(* CODESYS project ringbuffer.library
   Author: vscottki
   Placeholder: RingBuffer
   Title: RingBuffer
   Version: 1.4.0.999
   Company: Amazon

Project tree, tasks and I/O mapping:
  libraries: HelperFunctions, * (Amazon); Tc2_Standard, * (Beckhoff Automation GmbH); Tc2_System, * (Beckhoff Automation GmbH); Tc3_Module, * (Beckhoff Automation GmbH)
  DUTs/
    data type E_Divert
    data type ST_KeyValue
    data type ST_MoverDivert
    data type ST_RingBufferCfg
    data type ST_RingBufferStat
    data type ST_SystimeString
  GVLs/
    global variables Param_RingBuffer
  POUs/
    function block RingBufferBase [ST]: UpdateObjectCtInBuffers, P_ObjCountInBuffer, P_ObjectAdded, P_ObjectRemoved, ClearLastRemoved, IncrementPointer, UpdateAdded, UpdateIndices, UpdateRemoved, UpdateRemovePointer, UpdateWritePointer, FB_init
    function block RingBufferEventBase [ST]: ClearLastRemoved, UpdateRemovePointer, UpdateWritePointer, AddObjToBuffer, FB_init, P_LastObjectRemoved, RemoveObjFromBuffer, EqualsTo, EqualsToEventClass, EqualsToEventEntry, EqualsToEventEntryEx, eSeverity, EventClass, GetJsonAttribute, ipSourceInfo, nEventId, RequestEventClassName, RequestEventText, sEventClassName, sEventText, stEventEntry
    function block RingBufferKeyString [ST]: ClearLastRemoved, UpdateRemovePointer, UpdateWritePointer, AddObjToBuffer, FB_init, P_LastObjectRemoved, RemoveObjFromBuffer, CopyMemArea
    function block RingBufferMoverDivert [ST]: ClearLastRemoved, UpdateRemovePointer, UpdateWritePointer, AddObjToBuffer, FB_init, P_LastObjectRemoved, RemoveObjFromBuffer
    function UpdateKeyStrTimestamp [ST]
    function UpdateKeyValueTimestamp [ST]
  Project Information/
    function F_GetCompany [ST]
    function F_GetTitle [ST]
    function F_GetVersion [ST]
  Version/
    global variables Global_Version
  VISUs/
*)

// DUTs/E_Divert
{attribute 'qualified_only'}
{attribute 'strict'}
TYPE E_Divert :
(
	NoDivert := 0,
	Divert	:= 1
);
END_TYPE

// DUTs/ST_KeyValue
TYPE ST_KeyValue :
STRUCT
  key         : ULINT;    // system timestamp
  value       : ULINT; // SJsonValue;+ dynamically spool up instances of JSONDOMparser to create documents, then destroy them when completed; 
END_STRUCT
END_TYPE

// DUTs/ST_MoverDivert
TYPE ST_MoverDivert :
STRUCT
	MoverID						: UDINT;
	Divert						: E_Divert;
	DivertOnInterval	: BOOL;
	SysTime     			: ULINT;    // system timestamp
END_STRUCT
END_TYPE

// DUTs/ST_RingBufferCfg
TYPE ST_RingBufferCfg :
STRUCT
  CopyToLargeMemoryArea   : BOOL := TRUE;
  CopyOnlyUniqueMessage   : BOOL := FALSE;
  AllowOverwriteSecBuffer : BOOL := FALSE;
  ByteCountOfDataObj      : UDINT; // do not write to this manually; done using SIZEOF function
  WriteDataToFile         : BOOL := FALSE;
	RemoveAfterAdd					: BOOL;
END_STRUCT
END_TYPE

// DUTs/ST_RingBufferStat
TYPE ST_RingBufferStat :
STRUCT
  BufferIsFullPrim        : BOOL;
  BufferIsFullSec         : BOOL;  
  ObjectCountInBufferPrim : ULINT;
  ObjectCountInBufferSec  : ULINT;
  ObjectAddedPrimary      : BOOL;
  ObjectRemovedPrimary    : BOOL;
  ObjectAdded2ndary       : BOOL;
  ObjectRemoved2ndary     : BOOL;
  Overwriting             : BOOL;
  ByteCountInBufferPrim   : ULINT;  
  ByteCountInBufferSec    : ULINT;
  BufferCapacity          : UDINT;
END_STRUCT
END_TYPE

// DUTs/ST_SystimeString
TYPE ST_SystimeString :
STRUCT
  systimestamp   : ULINT;    // system timestamp
  sJson          : TcEventField.JsonAttribute;
  stringval      : Tc2_System.T_MaxString;
END_STRUCT
END_TYPE

// GVLs/Param_RingBuffer
{attribute 'qualified_only'}
VAR_GLOBAL CONSTANT
  MIN_NUMBER_OBJECTS : UDINT := 0;
  MAX_NUMBER_OBJECTS : UDINT := 4;
END_VAR

// Version/Global_Version
{attribute 'TcGenerated'}
{attribute 'no-analysis'}
{attribute 'linkalways'}
// This function has been automatically generated from the project information.
VAR_GLOBAL CONSTANT
	{attribute 'const_non_replaced'}
	stLibVersion_RingBuffer : ST_LibVersion := (iMajor := 1, iMinor := 4, iBuild := 0, iRevision := 999, nFlags := 0, sVersion := '1.4.0.999');
END_VAR

// POUs/RingBufferBase
FUNCTION_BLOCK ABSTRACT RingBufferBase
VAR
  RingBuffCfg             : ST_RingBufferCfg;
  pRemove                 : PVOID;
  pWrite                  : PVOID;
  pRemoveUpdated          : BOOL;
  pWriteUpdated           : BOOL;
  GlobalCounter           : UDINT;
  WriteIncrement          : UDINT;
  RemoveIncrement         : UDINT;
  WriteIndex              : UDINT;
  RemoveIndex             : UDINT;
  RingBufferStat          : ST_RingBufferStat;
END_VAR

UpdateObjectCtInBuffers();
UpdateIndices();

METHOD PRIVATE UpdateObjectCtInBuffers
IF RingBufferStat.ObjectAddedPrimary THEN
  IF GlobalCounter >= RingBufferStat.BufferCapacity THEN // In Buffer Overflow
    RingBufferStat.ObjectCountInBufferPrim   := RingBufferStat.BufferCapacity;
  ELSE
    RingBufferStat.ObjectCountInBufferPrim   := RingBufferStat.ObjectCountInBufferPrim +1;
	END_IF
END_IF

IF RingBufferStat.ObjectRemovedPrimary THEN
  RingBufferStat.ObjectCountInBufferPrim   := RingBufferStat.ObjectCountInBufferPrim -1; 
END_IF

//Primary - Ring
RingBufferStat.BufferIsFullPrim          := RingBufferStat.ObjectCountInBufferPrim = RingBufferStat.BufferCapacity;
                      
RingBufferStat.ByteCountInBufferPrim     := RingBufferStat.ObjectCountInBufferPrim * RingBuffCfg.ByteCountOfDataObj;

//Secondary
RingBufferStat.BufferIsFullSec           := RingBufferStat.ObjectCountInBufferSec = RingBufferStat.BufferCapacity;
                      
RingBufferStat.ByteCountInBufferSec      := RingBufferStat.ObjectCountInBufferSec * RingBuffCfg.ByteCountOfDataObj;
END_METHOD

{attribute 'monitoring' := 'call'}
PROPERTY P_ObjCountInBuffer : ULINT
GET
P_ObjCountInBuffer  := RingBufferStat.ObjectCountInBufferPrim;
END_GET
END_PROPERTY

PROPERTY P_ObjectAdded : REFERENCE TO BOOL
GET
P_ObjectAdded REF= RingBufferStat.ObjectAddedPrimary;
END_GET
END_PROPERTY

PROPERTY P_ObjectRemoved : REFERENCE TO BOOL
GET
P_ObjectRemoved REF= RingBufferStat.ObjectRemovedPrimary;
END_GET
END_PROPERTY

METHOD PROTECTED ABSTRACT ClearLastRemoved
END_METHOD

METHOD PROTECTED IncrementPointer : ULINT
VAR_INPUT
  pPointer        : PVOID;
  ByteCtIncrement : ULINT; 
END_VAR
IncrementPointer  := pPointer + ByteCtIncrement;
END_METHOD

METHOD PROTECTED UpdateAdded
IF RingBufferStat.ObjectAddedPrimary THEN
  RingBufferStat.ObjectAddedPrimary   := FALSE;
END_IF

IF RingBufferStat.ObjectAdded2ndary THEN
  RingBufferStat.ObjectAdded2ndary   := FALSE;
END_IF
END_METHOD

METHOD PROTECTED UpdateIndices
WriteIndex := (WriteIncrement MOD RingBufferStat.BufferCapacity) + Param_RingBuffer.MIN_NUMBER_OBJECTS;

IF GlobalCounter >= RingBufferStat.BufferCapacity THEN // Buffer Overflow
  RemoveIndex                 := WriteIndex+1;
  RingBufferStat.Overwriting  := TRUE;
ELSE
  RemoveIndex  := (RemoveIncrement MOD RingBufferStat.BufferCapacity) + Param_RingBuffer.MIN_NUMBER_OBJECTS;
  RingBufferStat.Overwriting  := FALSE;
END_IF
END_METHOD

METHOD PROTECTED UpdateRemoved
IF RingBufferStat.ObjectRemovedPrimary THEN
  RingBufferStat.ObjectRemovedPrimary   := FALSE;
END_IF

IF RingBufferStat.ObjectRemoved2ndary THEN
  RingBufferStat.ObjectRemoved2ndary   := FALSE;
END_IF
END_METHOD

METHOD PROTECTED ABSTRACT UpdateRemovePointer
VAR_INPUT
  pRemovePtr  : PVOID;
END_VAR
END_METHOD

METHOD PROTECTED ABSTRACT UpdateWritePointer
VAR_INPUT
  pWritePtr  : PVOID;
END_VAR
END_METHOD

METHOD FB_init : BOOL
VAR_INPUT
	bInitRetains : BOOL; // if TRUE, the retain variables are initialized (warm start / cold start)
	bInCopyCode : BOOL;  // if TRUE, the instance afterwards gets moved into the copy code (online change)
END_VAR
RingBufferStat.BufferCapacity  := (Param_RingBuffer.MAX_NUMBER_OBJECTS - Param_RingBuffer.MIN_NUMBER_OBJECTS) +1;
END_METHOD

END_FUNCTION_BLOCK

// POUs/RingBufferEventBase
FUNCTION_BLOCK RingBufferEventBase EXTENDS RingBufferBase
VAR
  Buffer              : ARRAY[Param_RingBuffer.MIN_NUMBER_OBJECTS..Param_RingBuffer.MAX_NUMBER_OBJECTS] 
                        OF ST_KeyValue;
//VAR_OUTPUT
  LastObjRemoved      : ST_KeyValue;
{warning 'Dependency injection from child FB?'}  
//  instQueryInterface  : I_Event := THIS^;//__SYSTEM.IQueryInterface;
END_VAR

SUPER^();

METHOD PROTECTED ClearLastRemoved
IF NOT pRemoveUpdated THEN
  MEMSET(destAddr := ADR(LastObjRemoved), fillByte := 16#00, n := RingBuffCfg.ByteCountOfDataObj);  
END_IF
END_METHOD

METHOD PROTECTED UpdateRemovePointer
VAR_INPUT
  pRemovePtr  : PVOID;
END_VAR
pRemove := ADR(Buffer[RemoveIndex]);

pRemoveUpdated  := TRUE;
END_METHOD

METHOD PROTECTED UpdateWritePointer
VAR_INPUT
  pWritePtr  : PVOID;
END_VAR
IF (WriteIndex = Param_RingBuffer.MIN_NUMBER_OBJECTS) THEN
  pWrite        := ADR(Buffer[Param_RingBuffer.MIN_NUMBER_OBJECTS]);
ELSIF (WriteIndex > Param_RingBuffer.MIN_NUMBER_OBJECTS) AND 
  (WriteIndex <= Param_RingBuffer.MAX_NUMBER_OBJECTS) THEN
  pWrite        := IncrementPointer(pPointer  := pWrite, ByteCtIncrement := RingBuffCfg.ByteCountOfDataObj);
END_IF

pWriteUpdated   := TRUE;
END_METHOD

METHOD PUBLIC AddObjToBuffer
VAR_INPUT
  RefObject           : REFERENCE TO ST_KeyValue;
END_VAR
VAR
  CountBytesWritten   : ULINT;
END_VAR
VAR_OUTPUT
  Error               : BOOL;
END_VAR
UpdateWritePointer(pWritePtr := pWrite);

IF __ISVALIDREF(RefObject) AND pWriteUpdated AND_THEN NOT pRemoveUpdated AND (GlobalCounter < 4294967295) THEN
  UpdateKeyValueTimestamp(DataObject := RefObject);
//  UpdateObjectMemLoc(DataObject := RefObject, _interface := instQueryInterface);
  CountBytesWritten := Tc2_System.MEMMOVE(srcAddr := ADR(RefObject), destAddr := pWrite, n := RingBuffCfg.ByteCountOfDataObj);
  pWriteUpdated     := FALSE;
{warning <'Check Global Buffer Overflow condition if Counter defined > MAX SIZE OF UDINT'>}
END_IF

IF (CountBytesWritten > 0) THEN
  GlobalCounter     := GlobalCounter +1;
  WriteIncrement    := WriteIncrement +1;
  RingBufferStat.ObjectAddedPrimary       := TRUE;
ELSIF (CountBytesWritten <= 0) THEN
  Error             := TRUE;
END_IF
END_METHOD

METHOD FB_init : BOOL
VAR_INPUT
	bInitRetains : BOOL; // if TRUE, the retain variables are initialized (warm start / cold start)
	bInCopyCode : BOOL;  // if TRUE, the instance afterwards gets moved into the copy code (online change)
END_VAR
RemoveIndex  := Param_RingBuffer.MIN_NUMBER_OBJECTS;

RingBuffCfg.ByteCountOfDataObj      := SIZEOF(Buffer[Param_RingBuffer.MIN_NUMBER_OBJECTS]);

IF (pWrite = Tc3_Module.NULL) THEN
  pWrite  := ADR(Buffer[Param_RingBuffer.MIN_NUMBER_OBJECTS]);
END_IF

IF (pRemove = Tc3_Module.NULL) THEN
  pRemove  := ADR(Buffer[Param_RingBuffer.MIN_NUMBER_OBJECTS]);
END_IF
END_METHOD

PROPERTY P_LastObjectRemoved : REFERENCE TO ST_KeyValue
GET
P_LastObjectRemoved REF= LastObjRemoved;
END_GET
END_PROPERTY

METHOD PUBLIC RemoveObjFromBuffer
VAR
  CountBytesRemoved  : ULINT;
  CountBytesCleared  : ULINT;  
END_VAR
VAR_OUTPUT
  Error              : BOOL;
END_VAR
UpdateRemovePointer(pRemovePtr := pRemove);

IF pRemoveUpdated AND_THEN NOT pWriteUpdated AND (GlobalCounter < 4294967295) THEN
  CountBytesRemoved := Tc2_System.MEMMOVE(srcAddr := pRemove, destAddr := ADR(LastObjRemoved), n := RingBuffCfg.ByteCountOfDataObj);
  pRemoveUpdated    := FALSE;
{warning <'Check Global Buffer Overflow condition'>}
{warning <'Create Check for IF pRemove = pWrite'>}
END_IF

IF (CountBytesRemoved > 0) AND (GlobalCounter >= 1) THEN
  CountBytesCleared := Tc2_System.MEMSET(destAddr := pRemove, fillByte := 16#00, n := RingBuffCfg.ByteCountOfDataObj);
  GlobalCounter     := GlobalCounter -1;
  RemoveIncrement   := RemoveIncrement +1;
  pRemove           := IncrementPointer(pPointer := pRemove, ByteCtIncrement := RingBuffCfg.ByteCountOfDataObj);
  RingBufferStat.ObjectRemovedPrimary     := TRUE;
ELSE
  Error             := TRUE;
END_IF

IF (CountBytesCleared > 0) THEN
//
ELSE
//  Error             := TRUE;
END_IF
END_METHOD

{warning 'add method implementation '}
(* returns TRUE if equal.*)
METHOD EqualsTo : BOOL
VAR_INPUT
	ipOther	: Tc3_EventLogger.I_TcEventBase;
END_VAR
END_METHOD

{warning 'add method implementation '}
(* returns TRUE if equal.*)
METHOD EqualsToEventClass : BOOL
VAR_INPUT
	OtherEventClass	: Tc3_EventLogger.GUID;
END_VAR
END_METHOD

{warning 'add method implementation '}
(* returns TRUE if equal.*)
METHOD EqualsToEventEntry : BOOL
VAR_INPUT
	OtherEventClass	: Tc3_EventLogger.GUID;
	nOtherEventID	: UDINT;
	eOtherSeverity	: Tc3_EventLogger.TcEventSeverity;
END_VAR
END_METHOD

{warning 'add method implementation '}
(* returns TRUE if equal.*)
METHOD EqualsToEventEntryEx : BOOL
VAR_INPUT
	stOther	: Tc3_EventLogger.TcEventEntry;
END_VAR
END_METHOD

{warning 'add property implementation'}
PROPERTY eSeverity : Tc3_EventLogger.TcEventSeverity
GET
END_GET
END_PROPERTY

{warning 'add property implementation'}
PROPERTY EventClass : Tc3_EventLogger.GUID
GET
END_GET
END_PROPERTY

{warning 'add method implementation '}
METHOD GetJsonAttribute : Tc3_EventLogger.HRESULT
VAR_INPUT
	sJsonAttribute	: REFERENCE TO STRING;
	nJsonAttribute	: UDINT;
END_VAR
END_METHOD

{warning 'add property implementation'}
PROPERTY ipSourceInfo : Tc3_EventLogger.I_TcSourceInfo
GET
END_GET
END_PROPERTY

{warning 'add property implementation'}
PROPERTY nEventId : UDINT
GET
END_GET
END_PROPERTY

{warning 'add method implementation '}
(* Async request for event text.
 Returns TRUE if async request is not any more busy.
 Result is only output if no error occurred.*)
METHOD RequestEventClassName : BOOL
VAR_INPUT
	(* English(US)=1033 ; German(Germay)=1031*)
	nLangId	: DINT;
	(* buffer for result text*)
	sResult	: REFERENCE TO STRING;
	(* size of buffer in bytes*)
	nResultSize	: UDINT;
END_VAR
VAR_OUTPUT
	bError	: BOOL;
	hrErrorCode	: Tc3_EventLogger.HRESULT;
END_VAR
END_METHOD

{warning 'add method implementation '}
(* Async request for event text.
 Returns TRUE if async request is not any more busy.
 Result is only output if no error occurred.*)
METHOD RequestEventText : BOOL
VAR_INPUT
	(* English(US)=1033 ; German(Germay)=1031*)
	nLangId	: DINT;
	(* buffer for result text*)
	sResult	: REFERENCE TO STRING;
	(* size of buffer in bytes*)
	nResultSize	: UDINT;
END_VAR
VAR_OUTPUT
	bError	: BOOL;
	hrErrorCode	: Tc3_EventLogger.HRESULT;
END_VAR
END_METHOD

{warning 'add property implementation'}
PROPERTY sEventClassName : STRING(255)
GET
END_GET
END_PROPERTY

{warning 'add property implementation'}
PROPERTY sEventText : STRING(255)
GET
END_GET
END_PROPERTY

{warning 'add property implementation'}
PROPERTY stEventEntry : Tc3_EventLogger.TcEventEntry
GET
END_GET
END_PROPERTY

END_FUNCTION_BLOCK

// POUs/UpdateKeyValueTimestamp
FUNCTION UpdateKeyValueTimestamp
VAR_IN_OUT
  DataObject        : ST_MoverDivert;
END_VAR

DataObject.SysTime        := SystemTimeUtcCorrected(HourDeltaUTC := Param_HelperFunctions.HourDeltaFromUtc);

END_FUNCTION

// POUs/RingBufferKeyString
FUNCTION_BLOCK RingBufferKeyString EXTENDS RingBufferBase
VAR
  Buffer              : ARRAY[Param_RingBuffer.MIN_NUMBER_OBJECTS..Param_RingBuffer.MAX_NUMBER_OBJECTS] 
                        OF ST_SystimeString;
//  StaticMemBuffer     : ARRAY[Param_RingBuffer.MIN_NUMBER_OBJECTS..Param_RingBuffer.MAX_NUMBER_OBJECTS] 
//                        OF ST_SystimeString;                       
//VAR_OUTPUT
  LastObjRemoved      : ST_SystimeString;
{warning 'Dependency injection from child FB?'}  
//  instQueryInterface  : I_Event := THIS^;//__SYSTEM.IQueryInterface;
END_VAR

CopyMemArea();

SUPER^();

METHOD PROTECTED ClearLastRemoved
IF NOT pRemoveUpdated THEN
  MEMSET(destAddr := ADR(LastObjRemoved), fillByte := 16#00, n := RingBuffCfg.ByteCountOfDataObj);  
END_IF
END_METHOD

METHOD PROTECTED UpdateRemovePointer
VAR_INPUT
  pRemovePtr  : PVOID;
END_VAR
pRemove := ADR(Buffer[RemoveIndex]);

pRemoveUpdated  := TRUE;
END_METHOD

METHOD PROTECTED UpdateWritePointer
VAR_INPUT
  pWritePtr  : PVOID;
END_VAR
IF (WriteIndex = Param_RingBuffer.MIN_NUMBER_OBJECTS) THEN
  pWrite        := ADR(Buffer[Param_RingBuffer.MIN_NUMBER_OBJECTS]);
ELSIF (WriteIndex > Param_RingBuffer.MIN_NUMBER_OBJECTS) AND 
  (WriteIndex <= Param_RingBuffer.MAX_NUMBER_OBJECTS) THEN
  pWrite        := IncrementPointer(pPointer  := pWrite, ByteCtIncrement := RingBuffCfg.ByteCountOfDataObj);
END_IF

pWriteUpdated   := TRUE;
END_METHOD

METHOD PUBLIC AddObjToBuffer
VAR_INPUT
  RefObject           : REFERENCE TO ST_SystimeString;
END_VAR
VAR
  CountBytesWritten   : ULINT;
END_VAR
VAR_OUTPUT
  Error               : BOOL;
END_VAR
UpdateWritePointer(pWritePtr := pWrite);

IF __ISVALIDREF(RefObject) AND pWriteUpdated AND_THEN NOT pRemoveUpdated AND (GlobalCounter < 4294967295) THEN
  UpdateKeyStrTimestamp(DataObject := RefObject);
//  UpdateObjectMemLoc(DataObject := RefObject, _interface := instQueryInterface);
  CountBytesWritten := Tc2_System.MEMMOVE(srcAddr := ADR(RefObject), destAddr := pWrite, n := RingBuffCfg.ByteCountOfDataObj);
  pWriteUpdated     := FALSE;
{warning <'Check Global Buffer Overflow condition if Counter defined > MAX SIZE OF UDINT'>}
END_IF

IF (CountBytesWritten > 0) THEN
  GlobalCounter     := GlobalCounter +1;
  WriteIncrement    := WriteIncrement +1;
  RingBufferStat.ObjectAddedPrimary       := TRUE;
ELSIF (CountBytesWritten <= 0) THEN
  Error             := TRUE;
END_IF
END_METHOD

METHOD FB_init : BOOL
VAR_INPUT
	bInitRetains : BOOL; // if TRUE, the retain variables are initialized (warm start / cold start)
	bInCopyCode : BOOL;  // if TRUE, the instance afterwards gets moved into the copy code (online change)
END_VAR
RemoveIndex  := Param_RingBuffer.MIN_NUMBER_OBJECTS;

RingBuffCfg.ByteCountOfDataObj      := SIZEOF(Buffer[Param_RingBuffer.MIN_NUMBER_OBJECTS]);

IF (pWrite = Tc3_Module.NULL) THEN
  pWrite  := ADR(Buffer[Param_RingBuffer.MIN_NUMBER_OBJECTS]);
END_IF

IF (pRemove = Tc3_Module.NULL) THEN
  pRemove  := ADR(Buffer[Param_RingBuffer.MIN_NUMBER_OBJECTS]);
END_IF
END_METHOD

PROPERTY P_LastObjectRemoved : REFERENCE TO ST_SystimeString
GET
P_LastObjectRemoved REF= LastObjRemoved;
END_GET
END_PROPERTY

METHOD PUBLIC RemoveObjFromBuffer
VAR
  CountBytesRemoved  : ULINT;
  CountBytesCleared  : ULINT;  
END_VAR
VAR_OUTPUT
  Error              : BOOL;
END_VAR
UpdateRemovePointer(pRemovePtr := pRemove);

IF pRemoveUpdated AND_THEN NOT pWriteUpdated AND (GlobalCounter < 4294967295) THEN
  CountBytesRemoved := Tc2_System.MEMMOVE(srcAddr := pRemove, destAddr := ADR(LastObjRemoved), n := RingBuffCfg.ByteCountOfDataObj);
  pRemoveUpdated    := FALSE;
{warning <'Check Global Buffer Overflow condition'>}
{warning <'Create Check for IF pRemove = pWrite'>}
END_IF

IF (CountBytesRemoved > 0) AND (GlobalCounter >= 1) THEN
  CountBytesCleared := Tc2_System.MEMSET(destAddr := pRemove, fillByte := 16#00, n := RingBuffCfg.ByteCountOfDataObj);
  GlobalCounter     := GlobalCounter -1;
  RemoveIncrement   := RemoveIncrement +1;
  pRemove           := IncrementPointer(pPointer := pRemove, ByteCtIncrement := RingBuffCfg.ByteCountOfDataObj);
  RingBufferStat.ObjectRemovedPrimary     := TRUE;
ELSE
  Error             := TRUE;
END_IF

IF (CountBytesCleared > 0) THEN
//
ELSE
//  Error             := TRUE;
END_IF
END_METHOD

METHOD PROTECTED CopyMemArea
VAR
  CountBytesCopiedPrimSec  : UDINT;
  CountBytesRemovedSec     : UDINT;
END_VAR
IF RingBuffCfg.CopyToLargeMemoryArea THEN
  IF SUPER^.RingBufferStat.ObjectCountInBufferPrim > 0 THEN
    RemoveObjFromBuffer();    
	END_IF
  IF SUPER^.RingBufferStat.ObjectRemovedPrimary THEN
    IF NOT SUPER^.RingBufferStat.Overwriting OR RingBuffCfg.AllowOverwriteSecBuffer THEN 
      CountBytesCopiedPrimSec  := Tc2_System.MEMCPY(srcAddr := ADR(LastObjRemoved), destAddr := ADR(StaticMemBuffer[SUPER^.RemoveIndex]), n := SIZEOF(LastObjRemoved));
    END_IF
	END_IF
END_IF

IF CountBytesCopiedPrimSec = RingBuffCfg.ByteCountOfDataObj THEN
  RingBufferStat.ObjectCountInBufferSec  := RingBufferStat.ObjectCountInBufferSec +1;
  ClearLastRemoved();
END_IF

IF RingBufferStat.BufferIsFullSec THEN
  IF RingBuffCfg.WriteDataToFile THEN
    //   CountBytesRemovedSec     := 
  ELSE
    CountBytesRemovedSec   := Tc2_System.MEMSET(destAddr := ADR(StaticMemBuffer[Param_RingBuffer.MIN_NUMBER_OBJECTS]), fillByte := 16#00, n := ULINT_TO_UDINT(RingBufferStat.ByteCountInBufferSec));
  END_IF
END_IF

IF CountBytesRemovedSec = RingBufferStat.BufferCapacity THEN
  RingBufferStat.ObjectCountInBufferSec := 0;
END_IF
END_METHOD

END_FUNCTION_BLOCK

// POUs/UpdateKeyStrTimestamp
FUNCTION UpdateKeyStrTimestamp
VAR_IN_OUT
  DataObject        : ST_SystimeString;
END_VAR

DataObject.systimestamp        := SystemTimeUtcCorrected(HourDeltaUTC := Param_HelperFunctions.HourDeltaFromUtc);

END_FUNCTION

// POUs/RingBufferMoverDivert
FUNCTION_BLOCK RingBufferMoverDivert EXTENDS RingBufferBase
VAR
  Buffer              : ARRAY[Param_RingBuffer.MIN_NUMBER_OBJECTS..Param_RingBuffer.MAX_NUMBER_OBJECTS] 
                        OF ST_MoverDivert;
//VAR_OUTPUT
  LastObjRemoved      : ST_MoverDivert;

END_VAR

SUPER^();

IF RingBuffCfg.RemoveAfterAdd THEN
	IF RingBufferStat.ObjectAddedPrimary THEN
		RemoveObjFromBuffer();
	END_IF
END_IF

UpdateAdded();
UpdateRemoved();

METHOD PROTECTED ClearLastRemoved
IF NOT pRemoveUpdated THEN
  MEMSET(destAddr := ADR(LastObjRemoved), fillByte := 16#00, n := RingBuffCfg.ByteCountOfDataObj);  
END_IF
END_METHOD

METHOD PROTECTED UpdateRemovePointer
VAR_INPUT
  pRemovePtr  : PVOID;
END_VAR
pRemove := ADR(Buffer[RemoveIndex]);

pRemoveUpdated  := TRUE;
END_METHOD

METHOD PROTECTED UpdateWritePointer
VAR_INPUT
  pWritePtr  : PVOID;
END_VAR
IF (WriteIndex = Param_RingBuffer.MIN_NUMBER_OBJECTS) THEN
  pWrite        := ADR(Buffer[Param_RingBuffer.MIN_NUMBER_OBJECTS]);
ELSIF (WriteIndex > Param_RingBuffer.MIN_NUMBER_OBJECTS) AND 
  (WriteIndex <= Param_RingBuffer.MAX_NUMBER_OBJECTS) THEN
  pWrite        := IncrementPointer(pPointer  := pWrite, ByteCtIncrement := RingBuffCfg.ByteCountOfDataObj);
END_IF

pWriteUpdated   := TRUE;
END_METHOD

METHOD PUBLIC AddObjToBuffer
VAR_INPUT
  RefObject           : REFERENCE TO ST_MoverDivert;
END_VAR
VAR
  CountBytesWritten   : ULINT;
END_VAR
VAR_OUTPUT
  Error               : BOOL;
END_VAR
UpdateWritePointer(pWritePtr := pWrite);

IF __ISVALIDREF(RefObject) AND pWriteUpdated AND_THEN NOT pRemoveUpdated AND (GlobalCounter < 4294967295) THEN
  UpdateKeyValueTimestamp(DataObject := RefObject);
//  UpdateObjectMemLoc(DataObject := RefObject, _interface := instQueryInterface);
  CountBytesWritten := Tc2_System.MEMMOVE(srcAddr := ADR(RefObject), destAddr := pWrite, n := RingBuffCfg.ByteCountOfDataObj);
  pWriteUpdated     := FALSE;
{warning <'Check Global Buffer Overflow condition if Counter defined > MAX SIZE OF UDINT'>}
END_IF

IF (CountBytesWritten > 0) THEN
  GlobalCounter     := GlobalCounter +1;
  WriteIncrement    := WriteIncrement +1;
  RingBufferStat.ObjectAddedPrimary       := TRUE;
ELSIF (CountBytesWritten <= 0) THEN
  Error             := TRUE;
END_IF
END_METHOD

METHOD FB_init : BOOL
VAR_INPUT
	bInitRetains : BOOL; // if TRUE, the retain variables are initialized (warm start / cold start)
	bInCopyCode : BOOL;  // if TRUE, the instance afterwards gets moved into the copy code (online change)
END_VAR
RemoveIndex  := Param_RingBuffer.MIN_NUMBER_OBJECTS;

RingBuffCfg.ByteCountOfDataObj      := SIZEOF(Buffer[Param_RingBuffer.MIN_NUMBER_OBJECTS]);

IF (pWrite = Tc3_Module.NULL) THEN
  pWrite  := ADR(Buffer[Param_RingBuffer.MIN_NUMBER_OBJECTS]);
END_IF

IF (pRemove = Tc3_Module.NULL) THEN
  pRemove  := ADR(Buffer[Param_RingBuffer.MIN_NUMBER_OBJECTS]);
END_IF
END_METHOD

PROPERTY P_LastObjectRemoved : REFERENCE TO ST_MoverDivert
GET
P_LastObjectRemoved REF= LastObjRemoved;
END_GET
END_PROPERTY

METHOD PUBLIC RemoveObjFromBuffer
VAR
  CountBytesRemoved  : ULINT;
  CountBytesCleared  : ULINT;  
END_VAR
VAR_OUTPUT
  Error              : BOOL;
END_VAR
UpdateRemovePointer(pRemovePtr := pRemove);

IF pRemoveUpdated AND_THEN NOT pWriteUpdated AND (GlobalCounter < 4294967295) THEN
  CountBytesRemoved := Tc2_System.MEMMOVE(srcAddr := pRemove, destAddr := ADR(LastObjRemoved), n := RingBuffCfg.ByteCountOfDataObj);
  pRemoveUpdated    := FALSE;
{warning <'Check Global Buffer Overflow condition'>}
{warning <'Create Check for IF pRemove = pWrite'>}
END_IF

IF (CountBytesRemoved > 0) AND (GlobalCounter >= 1) THEN
  CountBytesCleared := Tc2_System.MEMSET(destAddr := pRemove, fillByte := 16#00, n := RingBuffCfg.ByteCountOfDataObj);
  GlobalCounter     := GlobalCounter -1;
  RemoveIncrement   := RemoveIncrement +1;
  pRemove           := IncrementPointer(pPointer := pRemove, ByteCtIncrement := RingBuffCfg.ByteCountOfDataObj);
  RingBufferStat.ObjectRemovedPrimary     := TRUE;
ELSE
  Error             := TRUE;
END_IF

IF (CountBytesCleared > 0) THEN
//
ELSE
//  Error             := TRUE;
END_IF
END_METHOD

END_FUNCTION_BLOCK

// Project Information/F_GetCompany
// This function has been automatically generated from the project information.
{attribute 'signature_flag' := '1073741824'}
{attribute 'TcGenerated'}
{attribute 'no-analysis'}
FUNCTION F_GetCompany : WSTRING
VAR_INPUT
	
END_VAR

F_GetCompany := "Amazon";

END_FUNCTION

// Project Information/F_GetTitle
// This function has been automatically generated from the project information.
{attribute 'signature_flag' := '1073741824'}
{attribute 'TcGenerated'}
{attribute 'no-analysis'}
FUNCTION F_GetTitle : WSTRING
VAR_INPUT
	
END_VAR

F_GetTitle := "RingBuffer";

END_FUNCTION

// Project Information/F_GetVersion
// This function has been automatically generated from the project information.
{attribute 'signature_flag' := '1073741824'}
{attribute 'TcGenerated'}
{attribute 'no-analysis'}
FUNCTION F_GetVersion : ST_LibVersion
VAR_INPUT
	
END_VAR

F_GetVersion.iMajor := 1;
F_GetVersion.iMinor := 4;
F_GetVersion.iBuild := 0;
F_GetVersion.iRevision := 999;
F_GetVersion.sVersion := '1.4.0.999';
F_GetVersion.nFlags := 0;

END_FUNCTION
